PROGRAM P_Puls
VAR
	tonFlashOn			: 	TON;
	bFlashEnable			: 	BOOL;
	tonFlashOff			: 	TON;
END_VAR

tonFlashOn(IN:= bFlashEnable, PT:= t#1000ms);

IF	tonFlashOn.Q	THEN
	bFlashEnable	:= FALSE;
END_IF

tonFlashOff(IN:= NOT bFlashEnable, PT:= t#1000ms);

IF	tonFlashOff.Q	THEN
	bFlashEnable	:= TRUE;
END_IF

END_PROGRAM

(* stored: Version 1.1.0.1, ProductVersion 3.1.4024.15
   POU P_Puls: Id {c5ab2a54-7799-46fe-9e2e-e4f7e73115a1}, SpecialFunc None *)
